{attribute addProperty ShortName "CU010"}
{attribute addProperty Name "Controlled unit x_tempalte_x"}
FUNCTION_BLOCK CU010 EXTENDS CUBase 
VAR
    _cuProcessDataDisplay       :  CU010ProcessData := (Parent := THIS^);
    _cuTechnologicalDataDisplay :  CU010TechnologicalData := (Parent := THIS^);
    _components          		:  CU010Components := (Parent := THIS^);
	{attribute addProperty Name "<#MANUAL#>"}
    {attribute addProperty ToolTip "<#Start manual/Service mode#>"}	
    _manualTask : CU010ManualTask(THIS^);
	{attribute addProperty Name "<#GROUND#>"}
	{attribute addProperty ToolTip "<#Brings the device into basic position.#>"}
	_groundTask : CU010GroundTask(THIS^, TcoCore.eRestoreMode.None);
	{attribute addProperty Name "<#AUTOMAT#>"}
	{attribute addProperty ToolTip "<#Starts automatic sequence. Before start you need to perform grounding sequence.#>"}	
	_automatTask : CU010AutomatTask(THIS^, TcoCore.eRestoreMode.None);     
	{attribute addProperty Name "<#SUSPEND PROCESS#>"}
    {attribute addProperty ToolTip "<#Starts suspend sequence of process(automatic,ground sequence).#>"}	
    _suspendTask : CU010SuspendTask(THIS^, TcoCore.eRestoreMode.None);     
	{attribute addProperty Name "<#RECOVER PROCESS#>"}
    {attribute addProperty ToolTip "<#Starts suspend sequence of process(automatic,ground sequence).#>"}	
    _recoverTask : CU010RecoverTask(THIS^, TcoCore.eRestoreMode.None);     
END_VAR

THIS^.CuId := eStations.CU010;



(*
	This controlled unit's component initialization.
*)

THIS^.InitializeComponents();

(*
	This controlled unit process data crud operations handler.
	Control exchange of process data between this controlled unit and the data repository.
*)

_processData();
_productionPlaner();


(*
	
	Cu's Modes
	
*)

Automat();
Ground();
Manual();


_suspendTask();
_recoverTask();







(*
	When no mode is active 'Idle' method should be called.
	'NoMode' method shouls contain code that renders this cu idle. 
*)

IF NOT (AutomatTask.Task.Busy 
		OR GroundTask.Task.Busy
		OR ManualTask.Task.Busy) 
THEN
	Idle();
END_IF



(*
	Updates this controlled unit's information for the UI.
*)


UpdateInfo();

_cuProcessDataDisplay := ProcessDataManager.Data.CU010;
_cuTechnologicalDataDisplay := Technology.TechnologicalSettings.Data.CU010;

_settings.WarningCycleTime:= _cuTechnologicalDataDisplay.WarningCycleTime;
_settings.ErrorCycleTime:= _cuTechnologicalDataDisplay.ErrorCycleTime;
_settings.AnyRecurringFailure:= _cuTechnologicalDataDisplay.AnyRecurringFailure;
_settings.SameRecurringFailure:= _cuTechnologicalDataDisplay.SameRecurringFailure;

(*~
	<docu>
		<summary>
			Controls `automatic` mode of `CU010`.
		</summary>
	</docu>
~*)
METHOD Automat
VAR_INPUT
END_VAR
(*
	Enable condition to start `automatTask`.
	Modify according your needs.
	[! 
	THIS IS NOT SAFETY CONDITION. THE SAFETY OF PRESONNEL AND EQUIPMENT MUST BE ENSURED BY ADDITIONAL MEANS 
	TO COMPLY WITH REGULATIONS
	]
*)


//_automatTask.Task.Enabled := (_groundTask.GroundDone OR  _automatTask.Task.Busy) AND THIS^.Technology.AllowAutomat();

(*
	Invokes `groundTask` from technology object.
*)

//IF(Technology.AutomatAllTask.Execute()) THEN _automatTask.Task.Invoke(); END_IF;

//IF(Technology.ForceStepMode()) THEN
 //	_automatTask.ModeController.Mode := eSequencerMode.StepMode;
//END_IF 



(*
	or use default behavior from abstraction
*)
	SUPER^.Automat();

(*

	Executes sequence of automatic mode.

*)

_automatTask();
END_METHOD

PROPERTY AutomatTask : REFERENCE TO CUBaseAutomat
GET
AutomatTask REF= _automatTask;
END_GET
END_PROPERTY

PROPERTY Components : REFERENCE TO CU010Components
GET
Components REF= _components;
END_GET
END_PROPERTY

PROPERTY CuProcessData : REFERENCE TO CU010ProcessData
GET
CuProcessData ref=ProcessDataManager.Data.CU010;
END_GET
END_PROPERTY

(*~
	<docu>
		<summary>
			Controls `ground` mode of `CU010`.
		</summary>
	</docu>
~*)
METHOD Ground : BOOL
VAR_INPUT
END_VAR
(*
	Enable condition to start `groundTask`.
	Modify according your needs.
	[! 
	THIS IS NOT SAFETY CONDITION. THE SAFETY OF PRESONNEL AND EQUIPMENT MUST BE ENSURED BY ADDITIONAL MEANS 
	TO COMPLY WITH REGULATIONS
	]
*)

//_groundTask.Task.Enabled :=  THIS^.Technology.AllowGround();

(*
	Invokes `groundTask` from technology object.
*)

//IF(Technology.GroundAllTask.Execute()) THEN _groundTask.Task.Invoke(); END_IF;


//IF _groundTask.GroundDone AND _groundTask.Task.Execute() THEN _groundTask.Restore();_groundTask.Task.Invoke();END_IF;


(*
	or use default behavior from abstraction
*)
	SUPER^.Ground();




(*

	Executes sequence of groundTask.

*)

_groundTask();
END_METHOD

PROPERTY GroundTask : REFERENCE TO CUBaseGround
GET
GroundTask REF= _groundTask;
END_GET
END_PROPERTY

(*~
	<docu>
		<summary>
			Code to be called cylically when `CU010` idle; no other mode is active.
		</summary>
	</docu>
~*)
METHOD Idle : BOOL
END_METHOD

METHOD InitializeComponents : BOOL

VAR_INST
	tempBoolHome: BOOL;
	tempBoolWork: BOOL;
	tempBoolP4Home: BOOL;
	tempBoolP4Work: BOOL;
END_VAR

Components.PairTagTask();
Components.ReworkInstructionTask();
(*
components.Group1.horizontalCylinder(inoAtHomePos:=GVL_iXlinker.EC1.EK1200.IA1_EL1809.Channel_1.Input, 
							   inoAtWorkPos:=GVL_iXlinker.EC1.EK1200.IA1_EL1809.Channel_2.Input, 
							   inoToHomePos:=GVL_iXlinker.EC1.EK1200.IA1_EL1809.Channel_3.Input, 
							   inoToWorkPos:=GVL_iXlinker.EC1.EK1200.IA1_EL1809.Channel_4.Input);
Components.SingleAxis.Config.InfoTime:=T#4S;
Components.SingleAxis.Config.ErrorTime:=T#10S;



Components.SingleAxis(inEnable := ,
    inEnablePositive := ,
    inEnableNegative := ,
    inCalibrationCam := ,
    refAxis := GVL_iXlinker.Axis1,
	inoPositions:= _positions);
	
	

//Components.PickAndPlace();
//Components.PickAndPlace.Service();
		
Components.MultiAxis(inEnableAxis1 := ,
    inEnablePositiveAxis1 := ,
    inEnableNegativeAxis1 := ,
    inCalibrationCamAxis1 := ,
    refAxis1 := GVL_iXlinker.Axis1,
	inoPositions:= _positionsMulti);
	
			
//Components.PickAndPlace.Components.Manipulator(inEnableAxis1 := ,
//    inEnablePositiveAxis1 := ,
//    inEnableNegativeAxis1 := ,
//    inCalibrationCamAxis1 := ,
//    refAxis1 := GVL_iXlinker.Axis1,
//	inoPositions:= _positionsMulti);
*)

Components.PlsPaletizator.Components.I1_PresentBlisterEntry(inoSignal:=GVL_iXlinker.Ec.EC.EK.AB23.Channel_1.Input);
Components.PlsPaletizator.Components.I2_PresentBlisterEntryEmptySpace(inoSignal:=GVL_iXlinker.Ec.EC.Ek.AB23.Channel_2.Input);
Components.PlsPaletizator.Components.I3_PresentBlistersInBufferEmpty(inoSignal:=GVL_iXlinker.Ec.EC.Ek.AB23.Channel_3.Input);
Components.PlsPaletizator.Components.I4_PresentBlisterInWorkingPos(inoSignal:=GVL_iXlinker.Ec.EC.Ek.AB23.Channel_4.Input);
Components.PlsPaletizator.Components.I5_OutBlistersIsThrowedCorrectly(inoSignal:=GVL_iXlinker.Ec.EC.Ek.AB23.Channel_5.Input);
Components.PlsPaletizator.Components.I6_OutBlistersLisftSignal(inoSignal:=GVL_iXlinker.Ec.EC.Ek.AB23.Channel_6.Input);
Components.PlsPaletizator.Components.I7_OutBlistersIsAboveOutBuffer(inoSignal:=GVL_iXlinker.Ec.EC.Ek.AB23.Channel_7.Input);
Components.PlsPaletizator.Components.I8_OutBlistersBufferIsFull(inoSignal:=GVL_iXlinker.Ec.EC.Ek.AB23.Channel_8.Input);



Components.PlsPaletizator.Components.P1_VerticalSepareEntryBlisters
				(inoAtHomePos:=GVL_iXlinker.Ec.EC.Ek.AB21.Channel_1.Input,
				inoAtWorkPos:=GVL_iXlinker.Ec.EC.Ek.AB21.Channel_2.Input,
				inoToHomePos:=tempBoolHome,
				inoToWorkPos:=tempBoolWork);
GVL_iXlinker.Ec.EC.Ek.PNEU.Modules.Outputs.digital_Data_O[0].1:=tempBoolHome;
GVL_iXlinker.Ec.EC.Ek.PNEU.Modules.Outputs.digital_Data_O[0].0:=tempBoolWork;

Components.PlsPaletizator.Components.P2_VerticalSepareEntryBlisters
				(inoAtHomePos:=GVL_iXlinker.Ec.EC.Ek.AB21.Channel_3.Input,
				inoAtWorkPos:=GVL_iXlinker.Ec.EC.Ek.AB21.Channel_4.Input,
				inoToHomePos:=tempBoolHome,
				inoToWorkPos:=tempBoolWork);
GVL_iXlinker.Ec.EC.Ek.PNEU.Modules.Outputs.digital_Data_O[0].3:=tempBoolHome;
GVL_iXlinker.Ec.EC.Ek.PNEU.Modules.Outputs.digital_Data_O[0].2:=tempBoolWork;


Components.PlsPaletizator.Components.P3_HorizontalSepareEntryBlisters
				(inoAtHomePos1:=GVL_iXlinker.Ec.EC.Ek.AB21.Channel_5.Input,
				inoAtWorkPos1:=GVL_iXlinker.Ec.EC.Ek.AB21.Channel_6.Input,
				inoAtHomePos2:=GVL_iXlinker.Ec.EC.Ek.AB21.Channel_7.Input,
				inoAtWorkPos2:=GVL_iXlinker.Ec.EC.Ek.AB21.Channel_8.Input,
				inoToHomePos:=tempBoolHome,
				inoToWorkPos:=tempBoolWork);
GVL_iXlinker.Ec.EC.Ek.PNEU.Modules.Outputs.digital_Data_O[0].5:=tempBoolHome;
GVL_iXlinker.Ec.EC.Ek.PNEU.Modules.Outputs.digital_Data_O[0].4:=tempBoolWork;

Components.PlsPaletizator.Components.P4_FeedEntryBlister
				(inoAtHomePos:=GVL_iXlinker.Ec.EC.Ek.AB21.Channel_9.Input,
				inoAtWorkPos:=GVL_iXlinker.Ec.EC.Ek.AB21.Channel_10.Input,
				inoToHomePos:=tempBoolP4Home,
				inoToWorkPos:=tempBoolP4Work);
				

GVL_iXlinker.Ec.EC.Ek.PNEU.Modules.Outputs.digital_Data_O[0].7:=tempBoolP4Home;
GVL_iXlinker.Ec.EC.Ek.PNEU.Modules.Outputs.digital_Data_O[0].6:=tempBoolP4Work;

Components.PlsPaletizator.Components.P5_HorizontalSepareOutBlisters
				(inoAtHomePos1:=GVL_iXlinker.Ec.EC.Ek.AB21.Channel_11.Input,
				inoAtWorkPos1:=GVL_iXlinker.Ec.EC.Ek.AB21.Channel_12.Input,
				inoAtHomePos2:=GVL_iXlinker.Ec.EC.Ek.AB21.Channel_13.Input,
				inoAtWorkPos2:=GVL_iXlinker.Ec.EC.Ek.AB21.Channel_14.Input,
				inoToHomePos:=tempBoolHome,
				inoToWorkPos:=tempBoolWork);
GVL_iXlinker.Ec.EC.Ek.PNEU.Modules.Outputs.digital_Data_O[1].1:=tempBoolHome;
GVL_iXlinker.Ec.EC.Ek.PNEU.Modules.Outputs.digital_Data_O[1].0:=tempBoolWork;

Components.PlsPaletizator.Components.P6_VerticalSepareOutBlister
				(inoAtHomePos:=GVL_iXlinker.Ec.EC.Ek.AB21.Channel_15.Input,
				inoAtWorkPos:=GVL_iXlinker.Ec.EC.Ek.AB21.Channel_16.Input,
				inoToHomePos:=tempBoolHome,
				inoToWorkPos:=tempBoolWork);
GVL_iXlinker.Ec.EC.Ek.PNEU.Modules.Outputs.digital_Data_O[1].3:=tempBoolHome;
GVL_iXlinker.Ec.EC.Ek.PNEU.Modules.Outputs.digital_Data_O[1].2:=tempBoolWork;


Components.PlsPaletizator.Components.P7_SupportEntryBlister
				(inoAtHomePos:=GVL_iXlinker.Ec.EC.Ek.AB22.Channel_1.Input,
				inoAtWorkPos:=GVL_iXlinker.Ec.EC.Ek.AB22.Channel_2.Input,
				inoToHomePos:=tempBoolHome,
				inoToWorkPos:=tempBoolWork);
GVL_iXlinker.Ec.EC.Ek.PNEU.Modules.Outputs.digital_Data_O[2].1:=tempBoolHome;
GVL_iXlinker.Ec.EC.Ek.PNEU.Modules.Outputs.digital_Data_O[2].0:=tempBoolWork;

Components.PlsPaletizator.Components.P8_FixEntryBlisterSide
				(inoAtHomePos1:=GVL_iXlinker.Ec.EC.Ek.AB22.Channel_3.Input,
				inoAtWorkPos1:=GVL_iXlinker.Ec.EC.Ek.AB22.Channel_4.Input,
				inoAtHomePos2:=GVL_iXlinker.Ec.EC.Ek.AB22.Channel_5.Input,
				inoAtWorkPos2:=GVL_iXlinker.Ec.EC.Ek.AB22.Channel_6.Input,
				inoToHomePos:=tempBoolHome,
				inoToWorkPos:=tempBoolWork);
GVL_iXlinker.Ec.EC.Ek.PNEU.Modules.Outputs.digital_Data_O[2].3:=tempBoolHome;
GVL_iXlinker.Ec.EC.Ek.PNEU.Modules.Outputs.digital_Data_O[2].2:=tempBoolWork;

Components.PlsPaletizator(inSafeCondition:=GVL_iXlinker.Ec.EC.IA1.Channel_1.Input);
Components.PlsPaletizator.Service();
END_METHOD

(*~
	<docu>
		<summary>
			Controls `manual` mode of `CU010`.
		</summary>
	</docu>
~*)
METHOD Manual : BOOL
VAR_INPUT
END_VAR
(*
	Enable condition to start `automatTask`.
	Modify according your needs.
	[! 
	THIS IS NOT SAFETY CONDITION. THE SAFETY OF PRESONNEL AND EQUIPMENT MUST BE ENSURED BY ADDITIONAL MEANS 
	TO COMPLY WITH REGULATIONS
	]
*)

	//_manualTask.Task.Enabled := THIS^.Technology.AllowManual();

	
(*
	or use default behavior from abstraction
*)
	SUPER^.Manual();
	

(*

	Executes sequence of manualTask.

*)
_manualTask();
END_METHOD

PROPERTY ManualTask : REFERENCE TO TcoTaskedService
GET
ManualTask REF= _manualTask;
END_GET
END_PROPERTY

PROPERTY ProductionPlanerTask : REFERENCE TO ProductionPlaner
GET
ProductionPlanerTask REF= _productionPlaner;
END_GET
END_PROPERTY

PROPERTY RecoverTask : REFERENCE TO CUBaseRecover
GET
RecoverTask REF= _recoverTask;
END_GET
END_PROPERTY

PROPERTY StatusInfo : REFERENCE TO CUBaseStatusInfo
GET
StatusInfo ref= _statusInfo;
END_GET
END_PROPERTY

PROPERTY SuspendTask : REFERENCE TO CUBaseSuspend
GET
SuspendTask REF= _suspendTask;
END_GET
END_PROPERTY

PROPERTY Technology : REFERENCE TO Technology
GET
VAR
    _technology : POINTER TO Technology;
END_VAR
IF __QUERYPOINTER(Parent, _technology) THEN // Check if _Parent is Station001
    Technology REF= _technology^;              // If the check is successful dereference a pointer. simlar to THIS^ or SUPER^
END_IF
END_GET
END_PROPERTY

PROPERTY TechnologyData : REFERENCE TO CU010TechnologicalData
GET
TechnologyData ref=_cuTechnologicalDataDisplay;
END_GET
END_PROPERTY

END_FUNCTION_BLOCK

(* stored: Version 1.1.0.1
   POU CU010: Id {6b733187-dd58-4f2f-9875-70181d3f4553}, SpecialFunc None
   Folder Modes: Id {ee40f835-53b7-40be-a830-5deb32ffff30}
   Folder Tasks: Id {652480c1-efef-4d00-a795-f8dcdd6731b2}
   Method Automat: Id {627f49ba-8388-4b5f-be40-22141cef4369}
   Property AutomatTask: Id {f549b558-32e6-414c-a695-36be20b654fb}
   Get Get: Id {fd729f11-316f-4e95-9cdb-aa55fe1319b6}
   Property Components: Id {18d87891-e0ec-493b-b811-bc2054632ab1}
   Get Get: Id {d5dca6fe-9a74-4d4a-a090-8723bac17e5c}
   Property CuProcessData: Id {510eb3ae-9bf6-48f5-86d9-99e48c83b41a}
   Get Get: Id {0812c0d5-adbd-4d49-830e-7aac2f84bfde}
   Method Ground: Id {242b550c-f8d9-4e9a-994e-1d97702a6829}
   Property GroundTask: Id {7b6e22d3-e9fb-4dff-9d53-10932f8de2de}
   Get Get: Id {fbebe048-0a90-4b8d-b7fc-4cb4c8888789}
   Method Idle: Id {e8dcebc5-5096-4552-88d0-769ad5d47060}
   Method InitializeComponents: Id {120bfe11-9f89-44d6-8c16-d7231caed1f3}
   Method Manual: Id {31fe2517-057a-4f04-a773-7529f25a48d4}
   Property ManualTask: Id {679c68d7-c432-437a-93e3-5ec7baca4847}
   Get Get: Id {18066477-76cf-4f76-b867-5a68143966bb}
   Property ProductionPlanerTask: Id {b4493d96-3ecc-4e41-8165-34c0729909e5}
   Get Get: Id {49fb81ce-5d80-4798-8b03-dfdda9cd7f89}
   Property RecoverTask: Id {188759c6-923a-4b96-b2bc-dcfb00d3b1fc}
   Get Get: Id {e3d83b47-0cf1-47bf-a43e-726be585712f}
   Property StatusInfo: Id {28e503ca-0fd1-4e8d-b3b4-7289a90e4ad9}
   Get Get: Id {510ea2e5-d61c-4c1a-bda9-bb390f1378f4}
   Property SuspendTask: Id {0ee6361f-3a7e-44da-a285-5a4de1d78de5}
   Get Get: Id {9f9b3785-fc47-4b9f-ad48-27265d5f6148}
   Property Technology: Id {25d6f839-884f-4515-b2ce-e2c9c7e54000}
   Get Get: Id {f2022d0f-4a27-46cb-b5cc-56683f0af100}
   Property TechnologyData: Id {cb00ab3e-7b9b-4a75-8561-7a533dfb8ded}
   Get Get: Id {9eb27573-8c44-4bca-b715-cea7cee9aa0e} *)
